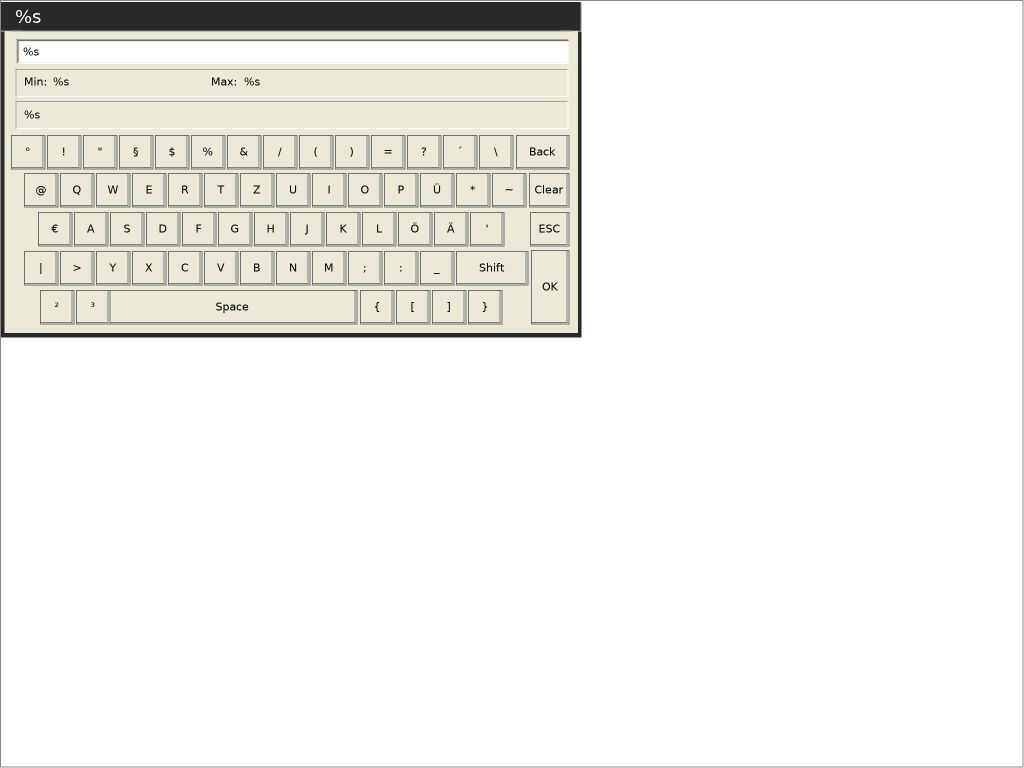
VISUALIZATION Keypad_Original  // 1024x768
VAR_INPUT
	stVariableValue : STRING;
	stMin : STRING;
	stMax : STRING;
	wstTitle : WSTRING;
	flags : DWORD;
END_VAR
VAR
	bInit : BOOL;
	bShift : BOOL := TRUE;
	stMessage : STRING;
	stOutputValue : STRING;
	iCaretPosition	: INT;
	iSelectionStart	: INT;
	iSelectionEnd	: INT;
	xAllSelected	: BOOL;
END_VAR
    Rectangle (2,28 578x40)
    Polyline (17,63) (17,39) (568,39)
    Polyline (18,63) (568,63) (568,40)
    Polyline (18,62) (18,40) (568,40)
    Textfield (20,42 547x20), "%s", text variable: stOutputValue
        p905179711: iCaretPosition
        p3815007873: iSelectionStart
        p1425650380: iSelectionEnd
        p3479897389: xAllSelected
    Rectangle (2,128 578x55)
    Rectangle (2,172 578x40)
    Rectangle (2,211 578x40)
    Rectangle (2,250 578x39)
    Rectangle (2,287 578x48)
    Button (531,250 38x74), "OK"
        OnMouseDown: CloseDialog Dialog=Keypad, Result=OK, NumpadKeypad=True, NumpadKeypadSet=True
    Button (530,212 39x34), "ESC"
        OnMouseDown: CloseDialog Dialog=Keypad, Result=Cancel, NumpadKeypad=True, NumpadKeypadSet=True
    Button (529,173 40x34), "Clear"
        OnMouseDown: execute {
            stVariableValue := '';
            stOutputValue := '';
            iCaretPosition	:= 1;
            iSelectionStart	:= 1;
            iSelectionEnd := 1;
        }
    Button (516,135 53x34), "Back"
        OnMouseDown: execute { VisuDlg_ProcessBack(stOutputValue, stVariableValue, iCaretPosition, iSelectionStart, iSelectionEnd, bInit); }
    Button (456,251 72x34), "Shift"
        OnMouseDown: toggle bShift
    Button (108,290 249x34), "Space"
        OnMouseDown: execute { VisuDlg_ProcessChar(stOutputValue, stVariableValue, iCaretPosition, iSelectionStart, iSelectionEnd, (flags AND VisuElems.Visu_InputFlags.Password) = 1, ' '); }
    Button (40,290 34x34), "²"
        OnMouseDown: execute { VisuDlg_ProcessChar(stOutputValue, stVariableValue, iCaretPosition, iSelectionStart, iSelectionEnd, (flags AND VisuElems.Visu_InputFlags.Password) = 1, '²'); }
    Button (76,290 34x34), "³"
        OnMouseDown: execute { VisuDlg_ProcessChar(stOutputValue, stVariableValue, iCaretPosition, iSelectionStart, iSelectionEnd, (flags AND VisuElems.Visu_InputFlags.Password) = 1, '³'); }
    Button (360,290 34x34), "{"
        OnMouseDown: execute { VisuDlg_ProcessChar(stOutputValue, stVariableValue, iCaretPosition, iSelectionStart, iSelectionEnd, (flags AND VisuElems.Visu_InputFlags.Password) = 1, '{'); }
    Button (396,290 34x34), "["
        OnMouseDown: execute { VisuDlg_ProcessChar(stOutputValue, stVariableValue, iCaretPosition, iSelectionStart, iSelectionEnd, (flags AND VisuElems.Visu_InputFlags.Password) = 1, '['); }
    Button (432,290 34x34), "]"
        OnMouseDown: execute { VisuDlg_ProcessChar(stOutputValue, stVariableValue, iCaretPosition, iSelectionStart, iSelectionEnd, (flags AND VisuElems.Visu_InputFlags.Password) = 1, ']'); }
    Button (468,290 34x34), "}"
        OnMouseDown: execute { VisuDlg_ProcessChar(stOutputValue, stVariableValue, iCaretPosition, iSelectionStart, iSelectionEnd, (flags AND VisuElems.Visu_InputFlags.Password) = 1, '}'); }
    Button (24,251 34x34), "|"
        OnMouseDown: execute { VisuDlg_ProcessChar(stOutputValue, stVariableValue, iCaretPosition, iSelectionStart, iSelectionEnd, (flags AND VisuElems.Visu_InputFlags.Password) = 1, '|'); }
    Button (60,251 34x34), "<", invisible if: NOT bShift
        OnMouseDown: execute { VisuDlg_ProcessChar(stOutputValue, stVariableValue, iCaretPosition, iSelectionStart, iSelectionEnd, (flags AND VisuElems.Visu_InputFlags.Password) = 1, '<'); }
    Button (60,251 34x34), ">", invisible if: bShift
        OnMouseDown: execute { VisuDlg_ProcessChar(stOutputValue, stVariableValue, iCaretPosition, iSelectionStart, iSelectionEnd, (flags AND VisuElems.Visu_InputFlags.Password) = 1, '>'); }
    Button (96,251 34x34), "y", invisible if: NOT bShift
        OnMouseDown: execute { VisuDlg_ProcessChar(stOutputValue, stVariableValue, iCaretPosition, iSelectionStart, iSelectionEnd, (flags AND VisuElems.Visu_InputFlags.Password) = 1, 'y'); }
    Button (96,251 34x34), "Y", invisible if: bShift
        OnMouseDown: execute { VisuDlg_ProcessChar(stOutputValue, stVariableValue, iCaretPosition, iSelectionStart, iSelectionEnd, (flags AND VisuElems.Visu_InputFlags.Password) = 1, 'Y'); }
    Button (132,251 34x34), "x", invisible if: NOT bShift
        OnMouseDown: execute { VisuDlg_ProcessChar(stOutputValue, stVariableValue, iCaretPosition, iSelectionStart, iSelectionEnd, (flags AND VisuElems.Visu_InputFlags.Password) = 1, 'x'); }
    Button (132,251 34x34), "X", invisible if: bShift
        OnMouseDown: execute { VisuDlg_ProcessChar(stOutputValue, stVariableValue, iCaretPosition, iSelectionStart, iSelectionEnd, (flags AND VisuElems.Visu_InputFlags.Password) = 1, 'X'); }
    Button (168,251 34x34), "c", invisible if: NOT bShift
        OnMouseDown: execute { VisuDlg_ProcessChar(stOutputValue, stVariableValue, iCaretPosition, iSelectionStart, iSelectionEnd, (flags AND VisuElems.Visu_InputFlags.Password) = 1, 'c'); }
    Button (168,251 34x34), "C", invisible if: bShift
        OnMouseDown: execute { VisuDlg_ProcessChar(stOutputValue, stVariableValue, iCaretPosition, iSelectionStart, iSelectionEnd, (flags AND VisuElems.Visu_InputFlags.Password) = 1, 'C'); }
    Button (204,251 34x34), "v", invisible if: NOT bShift
        OnMouseDown: execute { VisuDlg_ProcessChar(stOutputValue, stVariableValue, iCaretPosition, iSelectionStart, iSelectionEnd, (flags AND VisuElems.Visu_InputFlags.Password) = 1, 'v'); }
    Button (204,251 34x34), "V", invisible if: bShift
        OnMouseDown: execute { VisuDlg_ProcessChar(stOutputValue, stVariableValue, iCaretPosition, iSelectionStart, iSelectionEnd, (flags AND VisuElems.Visu_InputFlags.Password) = 1, 'V'); }
    Button (240,251 34x34), "b", invisible if: NOT bShift
        OnMouseDown: execute { VisuDlg_ProcessChar(stOutputValue, stVariableValue, iCaretPosition, iSelectionStart, iSelectionEnd, (flags AND VisuElems.Visu_InputFlags.Password) = 1, 'b'); }
    Button (240,251 34x34), "B", invisible if: bShift
        OnMouseDown: execute { VisuDlg_ProcessChar(stOutputValue, stVariableValue, iCaretPosition, iSelectionStart, iSelectionEnd, (flags AND VisuElems.Visu_InputFlags.Password) = 1, 'B'); }
    Button (276,251 34x34), "n", invisible if: NOT bShift
        OnMouseDown: execute { VisuDlg_ProcessChar(stOutputValue, stVariableValue, iCaretPosition, iSelectionStart, iSelectionEnd, (flags AND VisuElems.Visu_InputFlags.Password) = 1, 'n'); }
    Button (276,251 34x34), "N", invisible if: bShift
        OnMouseDown: execute { VisuDlg_ProcessChar(stOutputValue, stVariableValue, iCaretPosition, iSelectionStart, iSelectionEnd, (flags AND VisuElems.Visu_InputFlags.Password) = 1, 'N'); }
    Button (312,251 34x34), "m", invisible if: NOT bShift
        OnMouseDown: execute { VisuDlg_ProcessChar(stOutputValue, stVariableValue, iCaretPosition, iSelectionStart, iSelectionEnd, (flags AND VisuElems.Visu_InputFlags.Password) = 1, 'm'); }
    Button (312,251 34x34), "M", invisible if: bShift
        OnMouseDown: execute { VisuDlg_ProcessChar(stOutputValue, stVariableValue, iCaretPosition, iSelectionStart, iSelectionEnd, (flags AND VisuElems.Visu_InputFlags.Password) = 1, 'M'); }
    Button (348,251 34x34), ",", invisible if: NOT bShift
        OnMouseDown: execute { VisuDlg_ProcessChar(stOutputValue, stVariableValue, iCaretPosition, iSelectionStart, iSelectionEnd, (flags AND VisuElems.Visu_InputFlags.Password) = 1, ','); }
    Button (348,251 34x34), ";", invisible if: bShift
        OnMouseDown: execute { VisuDlg_ProcessChar(stOutputValue, stVariableValue, iCaretPosition, iSelectionStart, iSelectionEnd, (flags AND VisuElems.Visu_InputFlags.Password) = 1, ';'); }
    Button (384,251 34x34), ".", invisible if: NOT bShift
        OnMouseDown: execute { VisuDlg_ProcessChar(stOutputValue, stVariableValue, iCaretPosition, iSelectionStart, iSelectionEnd, (flags AND VisuElems.Visu_InputFlags.Password) = 1, '.'); }
    Button (384,251 34x34), ":", invisible if: bShift
        OnMouseDown: execute { VisuDlg_ProcessChar(stOutputValue, stVariableValue, iCaretPosition, iSelectionStart, iSelectionEnd, (flags AND VisuElems.Visu_InputFlags.Password) = 1, ':'); }
    Button (420,251 34x34), "-", invisible if: NOT bShift
        OnMouseDown: execute { VisuDlg_ProcessChar(stOutputValue, stVariableValue, iCaretPosition, iSelectionStart, iSelectionEnd, (flags AND VisuElems.Visu_InputFlags.Password) = 1, '-'); }
    Button (420,251 34x34), "_", invisible if: bShift
        OnMouseDown: execute { VisuDlg_ProcessChar(stOutputValue, stVariableValue, iCaretPosition, iSelectionStart, iSelectionEnd, (flags AND VisuElems.Visu_InputFlags.Password) = 1, '_'); }
    Button (38,212 34x34), "€"
        OnMouseDown: execute { VisuDlg_ProcessChar(stOutputValue, stVariableValue, iCaretPosition, iSelectionStart, iSelectionEnd, (flags AND VisuElems.Visu_InputFlags.Password) = 1, '€'); }
    Button (74,212 34x34), "a", invisible if: NOT bShift
        OnMouseDown: execute { VisuDlg_ProcessChar(stOutputValue, stVariableValue, iCaretPosition, iSelectionStart, iSelectionEnd, (flags AND VisuElems.Visu_InputFlags.Password) = 1, 'a'); }
    Button (74,212 34x34), "A", invisible if: bShift
        OnMouseDown: execute { VisuDlg_ProcessChar(stOutputValue, stVariableValue, iCaretPosition, iSelectionStart, iSelectionEnd, (flags AND VisuElems.Visu_InputFlags.Password) = 1, 'A'); }
    Button (110,212 34x34), "s", invisible if: NOT bShift
        OnMouseDown: execute { VisuDlg_ProcessChar(stOutputValue, stVariableValue, iCaretPosition, iSelectionStart, iSelectionEnd, (flags AND VisuElems.Visu_InputFlags.Password) = 1, 's'); }
    Button (110,212 34x34), "S", invisible if: bShift
        OnMouseDown: execute { VisuDlg_ProcessChar(stOutputValue, stVariableValue, iCaretPosition, iSelectionStart, iSelectionEnd, (flags AND VisuElems.Visu_InputFlags.Password) = 1, 'S'); }
    Button (146,212 34x34), "d", invisible if: NOT bShift
        OnMouseDown: execute { VisuDlg_ProcessChar(stOutputValue, stVariableValue, iCaretPosition, iSelectionStart, iSelectionEnd, (flags AND VisuElems.Visu_InputFlags.Password) = 1, 'd'); }
    Button (146,212 34x34), "D", invisible if: bShift
        OnMouseDown: execute { VisuDlg_ProcessChar(stOutputValue, stVariableValue, iCaretPosition, iSelectionStart, iSelectionEnd, (flags AND VisuElems.Visu_InputFlags.Password) = 1, 'D'); }
    Button (182,212 34x34), "f", invisible if: NOT bShift
        OnMouseDown: execute { VisuDlg_ProcessChar(stOutputValue, stVariableValue, iCaretPosition, iSelectionStart, iSelectionEnd, (flags AND VisuElems.Visu_InputFlags.Password) = 1, 'f'); }
    Button (182,212 34x34), "F", invisible if: bShift
        OnMouseDown: execute { VisuDlg_ProcessChar(stOutputValue, stVariableValue, iCaretPosition, iSelectionStart, iSelectionEnd, (flags AND VisuElems.Visu_InputFlags.Password) = 1, 'F'); }
    Button (218,212 34x34), "g", invisible if: NOT bShift
        OnMouseDown: execute { VisuDlg_ProcessChar(stOutputValue, stVariableValue, iCaretPosition, iSelectionStart, iSelectionEnd, (flags AND VisuElems.Visu_InputFlags.Password) = 1, 'g'); }
    Button (218,212 34x34), "G", invisible if: bShift
        OnMouseDown: execute { VisuDlg_ProcessChar(stOutputValue, stVariableValue, iCaretPosition, iSelectionStart, iSelectionEnd, (flags AND VisuElems.Visu_InputFlags.Password) = 1, 'G'); }
    Button (254,212 34x34), "h", invisible if: NOT bShift
        OnMouseDown: execute { VisuDlg_ProcessChar(stOutputValue, stVariableValue, iCaretPosition, iSelectionStart, iSelectionEnd, (flags AND VisuElems.Visu_InputFlags.Password) = 1, 'h'); }
    Button (254,212 34x34), "H", invisible if: bShift
        OnMouseDown: execute { VisuDlg_ProcessChar(stOutputValue, stVariableValue, iCaretPosition, iSelectionStart, iSelectionEnd, (flags AND VisuElems.Visu_InputFlags.Password) = 1, 'H'); }
    Button (290,212 34x34), "j", invisible if: NOT bShift
        OnMouseDown: execute { VisuDlg_ProcessChar(stOutputValue, stVariableValue, iCaretPosition, iSelectionStart, iSelectionEnd, (flags AND VisuElems.Visu_InputFlags.Password) = 1, 'j'); }
    Button (290,212 34x34), "J", invisible if: bShift
        OnMouseDown: execute { VisuDlg_ProcessChar(stOutputValue, stVariableValue, iCaretPosition, iSelectionStart, iSelectionEnd, (flags AND VisuElems.Visu_InputFlags.Password) = 1, 'J'); }
    Button (326,212 34x34), "k", invisible if: NOT bShift
        OnMouseDown: execute { VisuDlg_ProcessChar(stOutputValue, stVariableValue, iCaretPosition, iSelectionStart, iSelectionEnd, (flags AND VisuElems.Visu_InputFlags.Password) = 1, 'k'); }
    Button (326,212 34x34), "K", invisible if: bShift
        OnMouseDown: execute { VisuDlg_ProcessChar(stOutputValue, stVariableValue, iCaretPosition, iSelectionStart, iSelectionEnd, (flags AND VisuElems.Visu_InputFlags.Password) = 1, 'K'); }
    Button (362,212 34x34), "l", invisible if: NOT bShift
        OnMouseDown: execute { VisuDlg_ProcessChar(stOutputValue, stVariableValue, iCaretPosition, iSelectionStart, iSelectionEnd, (flags AND VisuElems.Visu_InputFlags.Password) = 1, 'l'); }
    Button (362,212 34x34), "L", invisible if: bShift
        OnMouseDown: execute { VisuDlg_ProcessChar(stOutputValue, stVariableValue, iCaretPosition, iSelectionStart, iSelectionEnd, (flags AND VisuElems.Visu_InputFlags.Password) = 1, 'L'); }
    Button (398,212 34x34), "ö", invisible if: NOT bShift
        OnMouseDown: execute { VisuDlg_ProcessChar(stOutputValue, stVariableValue, iCaretPosition, iSelectionStart, iSelectionEnd, (flags AND VisuElems.Visu_InputFlags.Password) = 1, 'ö'); }
    Button (398,212 34x34), "Ö", invisible if: bShift
        OnMouseDown: execute { VisuDlg_ProcessChar(stOutputValue, stVariableValue, iCaretPosition, iSelectionStart, iSelectionEnd, (flags AND VisuElems.Visu_InputFlags.Password) = 1, 'Ö'); }
    Button (434,212 34x34), "ä", invisible if: NOT bShift
        OnMouseDown: execute { VisuDlg_ProcessChar(stOutputValue, stVariableValue, iCaretPosition, iSelectionStart, iSelectionEnd, (flags AND VisuElems.Visu_InputFlags.Password) = 1, 'ä'); }
    Button (434,212 34x34), "Ä", invisible if: bShift
        OnMouseDown: execute { VisuDlg_ProcessChar(stOutputValue, stVariableValue, iCaretPosition, iSelectionStart, iSelectionEnd, (flags AND VisuElems.Visu_InputFlags.Password) = 1, 'Ä'); }
    Button (470,212 34x34), "#", invisible if: NOT bShift
        OnMouseDown: execute { VisuDlg_ProcessChar(stOutputValue, stVariableValue, iCaretPosition, iSelectionStart, iSelectionEnd, (flags AND VisuElems.Visu_InputFlags.Password) = 1, '#'); }
    Button (470,212 34x34), "'", invisible if: bShift
        OnMouseDown: execute { VisuDlg_ProcessChar(stOutputValue, stVariableValue, iCaretPosition, iSelectionStart, iSelectionEnd, (flags AND VisuElems.Visu_InputFlags.Password) = 1, '$''); }
    Button (24,173 34x34), "@"
        OnMouseDown: execute { VisuDlg_ProcessChar(stOutputValue, stVariableValue, iCaretPosition, iSelectionStart, iSelectionEnd, (flags AND VisuElems.Visu_InputFlags.Password) = 1, '@'); }
    Button (60,173 34x34), "q", invisible if: NOT bShift
        OnMouseDown: execute { VisuDlg_ProcessChar(stOutputValue, stVariableValue, iCaretPosition, iSelectionStart, iSelectionEnd, (flags AND VisuElems.Visu_InputFlags.Password) = 1, 'q'); }
    Button (60,173 34x34), "Q", invisible if: bShift
        OnMouseDown: execute { VisuDlg_ProcessChar(stOutputValue, stVariableValue, iCaretPosition, iSelectionStart, iSelectionEnd, (flags AND VisuElems.Visu_InputFlags.Password) = 1, 'Q'); }
    Button (96,173 34x34), "w", invisible if: NOT bShift
        OnMouseDown: execute { VisuDlg_ProcessChar(stOutputValue, stVariableValue, iCaretPosition, iSelectionStart, iSelectionEnd, (flags AND VisuElems.Visu_InputFlags.Password) = 1, 'w'); }
    Button (96,173 34x34), "W", invisible if: bShift
        OnMouseDown: execute { VisuDlg_ProcessChar(stOutputValue, stVariableValue, iCaretPosition, iSelectionStart, iSelectionEnd, (flags AND VisuElems.Visu_InputFlags.Password) = 1, 'W'); }
    Button (132,173 34x34), "e", invisible if: NOT bShift
        OnMouseDown: execute { VisuDlg_ProcessChar(stOutputValue, stVariableValue, iCaretPosition, iSelectionStart, iSelectionEnd, (flags AND VisuElems.Visu_InputFlags.Password) = 1, 'e'); }
    Button (132,173 34x34), "E", invisible if: bShift
        OnMouseDown: execute { VisuDlg_ProcessChar(stOutputValue, stVariableValue, iCaretPosition, iSelectionStart, iSelectionEnd, (flags AND VisuElems.Visu_InputFlags.Password) = 1, 'E'); }
    Button (168,173 34x34), "r", invisible if: NOT bShift
        OnMouseDown: execute { VisuDlg_ProcessChar(stOutputValue, stVariableValue, iCaretPosition, iSelectionStart, iSelectionEnd, (flags AND VisuElems.Visu_InputFlags.Password) = 1, 'r'); }
    Button (168,173 34x34), "R", invisible if: bShift
        OnMouseDown: execute { VisuDlg_ProcessChar(stOutputValue, stVariableValue, iCaretPosition, iSelectionStart, iSelectionEnd, (flags AND VisuElems.Visu_InputFlags.Password) = 1, 'R'); }
    Button (204,173 34x34), "t", invisible if: NOT bShift
        OnMouseDown: execute { VisuDlg_ProcessChar(stOutputValue, stVariableValue, iCaretPosition, iSelectionStart, iSelectionEnd, (flags AND VisuElems.Visu_InputFlags.Password) = 1, 't'); }
    Button (204,173 34x34), "T", invisible if: bShift
        OnMouseDown: execute { VisuDlg_ProcessChar(stOutputValue, stVariableValue, iCaretPosition, iSelectionStart, iSelectionEnd, (flags AND VisuElems.Visu_InputFlags.Password) = 1, 'T'); }
    Button (240,173 34x34), "z", invisible if: NOT bShift
        OnMouseDown: execute { VisuDlg_ProcessChar(stOutputValue, stVariableValue, iCaretPosition, iSelectionStart, iSelectionEnd, (flags AND VisuElems.Visu_InputFlags.Password) = 1, 'z'); }
    Button (240,173 34x34), "Z", invisible if: bShift
        OnMouseDown: execute { VisuDlg_ProcessChar(stOutputValue, stVariableValue, iCaretPosition, iSelectionStart, iSelectionEnd, (flags AND VisuElems.Visu_InputFlags.Password) = 1, 'Z'); }
    Button (276,173 34x34), "u", invisible if: NOT bShift
        OnMouseDown: execute { VisuDlg_ProcessChar(stOutputValue, stVariableValue, iCaretPosition, iSelectionStart, iSelectionEnd, (flags AND VisuElems.Visu_InputFlags.Password) = 1, 'u'); }
    Button (276,173 34x34), "U", invisible if: bShift
        OnMouseDown: execute { VisuDlg_ProcessChar(stOutputValue, stVariableValue, iCaretPosition, iSelectionStart, iSelectionEnd, (flags AND VisuElems.Visu_InputFlags.Password) = 1, 'U'); }
    Button (312,173 34x34), "i", invisible if: NOT bShift
        OnMouseDown: execute { VisuDlg_ProcessChar(stOutputValue, stVariableValue, iCaretPosition, iSelectionStart, iSelectionEnd, (flags AND VisuElems.Visu_InputFlags.Password) = 1, 'i'); }
    Button (312,173 34x34), "I", invisible if: bShift
        OnMouseDown: execute { VisuDlg_ProcessChar(stOutputValue, stVariableValue, iCaretPosition, iSelectionStart, iSelectionEnd, (flags AND VisuElems.Visu_InputFlags.Password) = 1, 'I'); }
    Button (348,173 34x34), "o", invisible if: NOT bShift
        OnMouseDown: execute { VisuDlg_ProcessChar(stOutputValue, stVariableValue, iCaretPosition, iSelectionStart, iSelectionEnd, (flags AND VisuElems.Visu_InputFlags.Password) = 1, 'o'); }
    Button (348,173 34x34), "O", invisible if: bShift
        OnMouseDown: execute { VisuDlg_ProcessChar(stOutputValue, stVariableValue, iCaretPosition, iSelectionStart, iSelectionEnd, (flags AND VisuElems.Visu_InputFlags.Password) = 1, 'O'); }
    Button (384,173 34x34), "p", invisible if: NOT bShift
        OnMouseDown: execute { VisuDlg_ProcessChar(stOutputValue, stVariableValue, iCaretPosition, iSelectionStart, iSelectionEnd, (flags AND VisuElems.Visu_InputFlags.Password) = 1, 'p'); }
    Button (384,173 34x34), "P", invisible if: bShift
        OnMouseDown: execute { VisuDlg_ProcessChar(stOutputValue, stVariableValue, iCaretPosition, iSelectionStart, iSelectionEnd, (flags AND VisuElems.Visu_InputFlags.Password) = 1, 'P'); }
    Button (420,173 34x34), "ü", invisible if: NOT bShift
        OnMouseDown: execute { VisuDlg_ProcessChar(stOutputValue, stVariableValue, iCaretPosition, iSelectionStart, iSelectionEnd, (flags AND VisuElems.Visu_InputFlags.Password) = 1, 'ü'); }
    Button (420,173 34x34), "Ü", invisible if: bShift
        OnMouseDown: execute { VisuDlg_ProcessChar(stOutputValue, stVariableValue, iCaretPosition, iSelectionStart, iSelectionEnd, (flags AND VisuElems.Visu_InputFlags.Password) = 1, 'Ü'); }
    Button (456,173 34x34), "+", invisible if: NOT bShift
        OnMouseDown: execute { VisuDlg_ProcessChar(stOutputValue, stVariableValue, iCaretPosition, iSelectionStart, iSelectionEnd, (flags AND VisuElems.Visu_InputFlags.Password) = 1, '+'); }
    Button (456,173 34x34), "*", invisible if: bShift
        OnMouseDown: execute { VisuDlg_ProcessChar(stOutputValue, stVariableValue, iCaretPosition, iSelectionStart, iSelectionEnd, (flags AND VisuElems.Visu_InputFlags.Password) = 1, '*'); }
    Button (492,173 34x34), "~"
        OnMouseDown: execute { VisuDlg_ProcessChar(stOutputValue, stVariableValue, iCaretPosition, iSelectionStart, iSelectionEnd, (flags AND VisuElems.Visu_InputFlags.Password) = 1, '~'); }
    Button (11,135 34x34), "^", invisible if: NOT bShift
        OnMouseDown: execute { VisuDlg_ProcessChar(stOutputValue, stVariableValue, iCaretPosition, iSelectionStart, iSelectionEnd, (flags AND VisuElems.Visu_InputFlags.Password) = 1, '^'); }
    Button (11,135 34x34), "°", invisible if: bShift
        OnMouseDown: execute { VisuDlg_ProcessChar(stOutputValue, stVariableValue, iCaretPosition, iSelectionStart, iSelectionEnd, (flags AND VisuElems.Visu_InputFlags.Password) = 1, '°'); }
    Button (47,135 34x34), "1", invisible if: NOT bShift
        OnMouseDown: execute { VisuDlg_ProcessChar(stOutputValue, stVariableValue, iCaretPosition, iSelectionStart, iSelectionEnd, (flags AND VisuElems.Visu_InputFlags.Password) = 1, '1'); }
    Button (47,135 34x34), "!", invisible if: bShift
        OnMouseDown: execute { VisuDlg_ProcessChar(stOutputValue, stVariableValue, iCaretPosition, iSelectionStart, iSelectionEnd, (flags AND VisuElems.Visu_InputFlags.Password) = 1, '!'); }
    Button (83,135 34x34), "2", invisible if: NOT bShift
        OnMouseDown: execute { VisuDlg_ProcessChar(stOutputValue, stVariableValue, iCaretPosition, iSelectionStart, iSelectionEnd, (flags AND VisuElems.Visu_InputFlags.Password) = 1, '2'); }
    Button (83,135 34x34), """, invisible if: bShift
        OnMouseDown: execute { VisuDlg_ProcessChar(stOutputValue, stVariableValue, iCaretPosition, iSelectionStart, iSelectionEnd, (flags AND VisuElems.Visu_InputFlags.Password) = 1, '"'); }
    Button (119,135 34x34), "3", invisible if: NOT bShift
        OnMouseDown: execute { VisuDlg_ProcessChar(stOutputValue, stVariableValue, iCaretPosition, iSelectionStart, iSelectionEnd, (flags AND VisuElems.Visu_InputFlags.Password) = 1, '3'); }
    Button (119,135 34x34), "§", invisible if: bShift
        OnMouseDown: execute { VisuDlg_ProcessChar(stOutputValue, stVariableValue, iCaretPosition, iSelectionStart, iSelectionEnd, (flags AND VisuElems.Visu_InputFlags.Password) = 1, '§'); }
    Button (155,135 34x34), "4", invisible if: NOT bShift
        OnMouseDown: execute { VisuDlg_ProcessChar(stOutputValue, stVariableValue, iCaretPosition, iSelectionStart, iSelectionEnd, (flags AND VisuElems.Visu_InputFlags.Password) = 1, '4'); }
    Button (155,135 34x34), "$", invisible if: bShift
        OnMouseDown: execute { VisuDlg_ProcessChar(stOutputValue, stVariableValue, iCaretPosition, iSelectionStart, iSelectionEnd, (flags AND VisuElems.Visu_InputFlags.Password) = 1, '$$'); }
    Button (191,135 34x34), "5", invisible if: NOT bShift
        OnMouseDown: execute { VisuDlg_ProcessChar(stOutputValue, stVariableValue, iCaretPosition, iSelectionStart, iSelectionEnd, (flags AND VisuElems.Visu_InputFlags.Password) = 1, '5'); }
    Button (191,135 34x34), "%", invisible if: bShift
        OnMouseDown: execute { VisuDlg_ProcessChar(stOutputValue, stVariableValue, iCaretPosition, iSelectionStart, iSelectionEnd, (flags AND VisuElems.Visu_InputFlags.Password) = 1, '%'); }
    Button (227,135 34x34), "6", invisible if: NOT bShift
        OnMouseDown: execute { VisuDlg_ProcessChar(stOutputValue, stVariableValue, iCaretPosition, iSelectionStart, iSelectionEnd, (flags AND VisuElems.Visu_InputFlags.Password) = 1, '6'); }
    Button (227,135 34x34), "&", invisible if: bShift
        OnMouseDown: execute { VisuDlg_ProcessChar(stOutputValue, stVariableValue, iCaretPosition, iSelectionStart, iSelectionEnd, (flags AND VisuElems.Visu_InputFlags.Password) = 1, '&'); }
    Button (263,135 34x34), "7", invisible if: NOT bShift
        OnMouseDown: execute { VisuDlg_ProcessChar(stOutputValue, stVariableValue, iCaretPosition, iSelectionStart, iSelectionEnd, (flags AND VisuElems.Visu_InputFlags.Password) = 1, '7'); }
    Button (263,135 34x34), "/", invisible if: bShift
        OnMouseDown: execute { VisuDlg_ProcessChar(stOutputValue, stVariableValue, iCaretPosition, iSelectionStart, iSelectionEnd, (flags AND VisuElems.Visu_InputFlags.Password) = 1, '/'); }
    Button (299,135 34x34), "8", invisible if: NOT bShift
        OnMouseDown: execute { VisuDlg_ProcessChar(stOutputValue, stVariableValue, iCaretPosition, iSelectionStart, iSelectionEnd, (flags AND VisuElems.Visu_InputFlags.Password) = 1, '8'); }
    Button (299,135 34x34), "(", invisible if: bShift
        OnMouseDown: execute { VisuDlg_ProcessChar(stOutputValue, stVariableValue, iCaretPosition, iSelectionStart, iSelectionEnd, (flags AND VisuElems.Visu_InputFlags.Password) = 1, '('); }
    Button (335,135 34x34), "9", invisible if: NOT bShift
        OnMouseDown: execute { VisuDlg_ProcessChar(stOutputValue, stVariableValue, iCaretPosition, iSelectionStart, iSelectionEnd, (flags AND VisuElems.Visu_InputFlags.Password) = 1, '9'); }
    Button (335,135 34x34), ")", invisible if: bShift
        OnMouseDown: execute { VisuDlg_ProcessChar(stOutputValue, stVariableValue, iCaretPosition, iSelectionStart, iSelectionEnd, (flags AND VisuElems.Visu_InputFlags.Password) = 1, ')'); }
    Button (371,135 34x34), "0", invisible if: NOT bShift
        OnMouseDown: execute { VisuDlg_ProcessChar(stOutputValue, stVariableValue, iCaretPosition, iSelectionStart, iSelectionEnd, (flags AND VisuElems.Visu_InputFlags.Password) = 1, '0'); }
    Button (371,135 34x34), "=", invisible if: bShift
        OnMouseDown: execute { VisuDlg_ProcessChar(stOutputValue, stVariableValue, iCaretPosition, iSelectionStart, iSelectionEnd, (flags AND VisuElems.Visu_InputFlags.Password) = 1, '='); }
    Button (407,135 34x34), "ß", invisible if: NOT bShift
        OnMouseDown: execute { VisuDlg_ProcessChar(stOutputValue, stVariableValue, iCaretPosition, iSelectionStart, iSelectionEnd, (flags AND VisuElems.Visu_InputFlags.Password) = 1, 'ß'); }
    Button (407,135 34x34), "?", invisible if: bShift
        OnMouseDown: execute { VisuDlg_ProcessChar(stOutputValue, stVariableValue, iCaretPosition, iSelectionStart, iSelectionEnd, (flags AND VisuElems.Visu_InputFlags.Password) = 1, '?'); }
    Button (443,135 34x34), "´"
        OnMouseDown: execute { VisuDlg_ProcessChar(stOutputValue, stVariableValue, iCaretPosition, iSelectionStart, iSelectionEnd, (flags AND VisuElems.Visu_InputFlags.Password) = 1, '´'); }
    Button (479,135 34x34), "\"
        OnMouseDown: execute { VisuDlg_ProcessChar(stOutputValue, stVariableValue, iCaretPosition, iSelectionStart, iSelectionEnd, (flags AND VisuElems.Visu_InputFlags.Password) = 1, '\'); }
    Rectangle (2,67 578x62)
    Rectangle (21,105 546x20), "%s", text variable: stMessage
    Rectangle (578,2 3x332)
    Rectangle (1,2 3x332)
    Rectangle (1,333 580x4)
    Polyline (16,128) (16,101) (568,101)
    Polyline (16,96) (16,69) (568,69)
    Polyline (17,128) (568,128) (568,101)
    Polyline (17,96) (568,96) (568,69)
    Image (1,2 580x29), image: Title2
    Rectangle (1,2 579x28), invisible if: VisuElems.g_VisualizationStyle.GetDINT('Dialog-UseHeaderColor', 0, 0) = 0
    Rectangle (12,7 563x20), "%s", text variable: wstTitle
    Rectangle (21,72 31x20), "Min:", invisible if: LEN(stMin) = 0
        p55702900: SEL(((UDINT_TO_DINT(flags AND 16#008))=16#0010),16#FF000000,16#FFFF0000)
    Rectangle (50,72 95x20), "%s", text variable: stMin, invisible if: LEN(stMin) = 0
        p55702900: SEL(((UDINT_TO_DINT(flags AND 16#0010))=16#0010),16#FF000000,16#FFFF0000)
    Rectangle (208,72 31x20), "Max:", invisible if: LEN(stMax) = 0
        p55702900: SEL(((UDINT_TO_DINT(flags AND 16#0010))=16#0010),16#FF000000,16#FFFF0000)
    Rectangle (241,72 95x20), "%s", text variable: stMax, invisible if: LEN(stMax) = 0
        p55702900: SEL(((UDINT_TO_DINT(flags AND 16#0010))=16#0010),16#FF000000,16#FFFF0000)
END_VISUALIZATION

(* stored: Version 1.1.0.1, ProductVersion 3.1.4024.2
   Visu Keypad_Original: Id {6504c4c4-334d-4760-9118-966df1ecf594} *)
